FUNCTION_BLOCK FB_Fenster_Logik
VAR_IN_OUT
	Steuerung	: ST_Fenster_Steuerung;
	Zustand		: ST_Fenster_Zustand;
END_VAR
VAR_INPUT
	Parameter	: ST_Fenster_Parameter;
END_VAR
VAR_OUTPUT
END_VAR
VAR
END_VAR

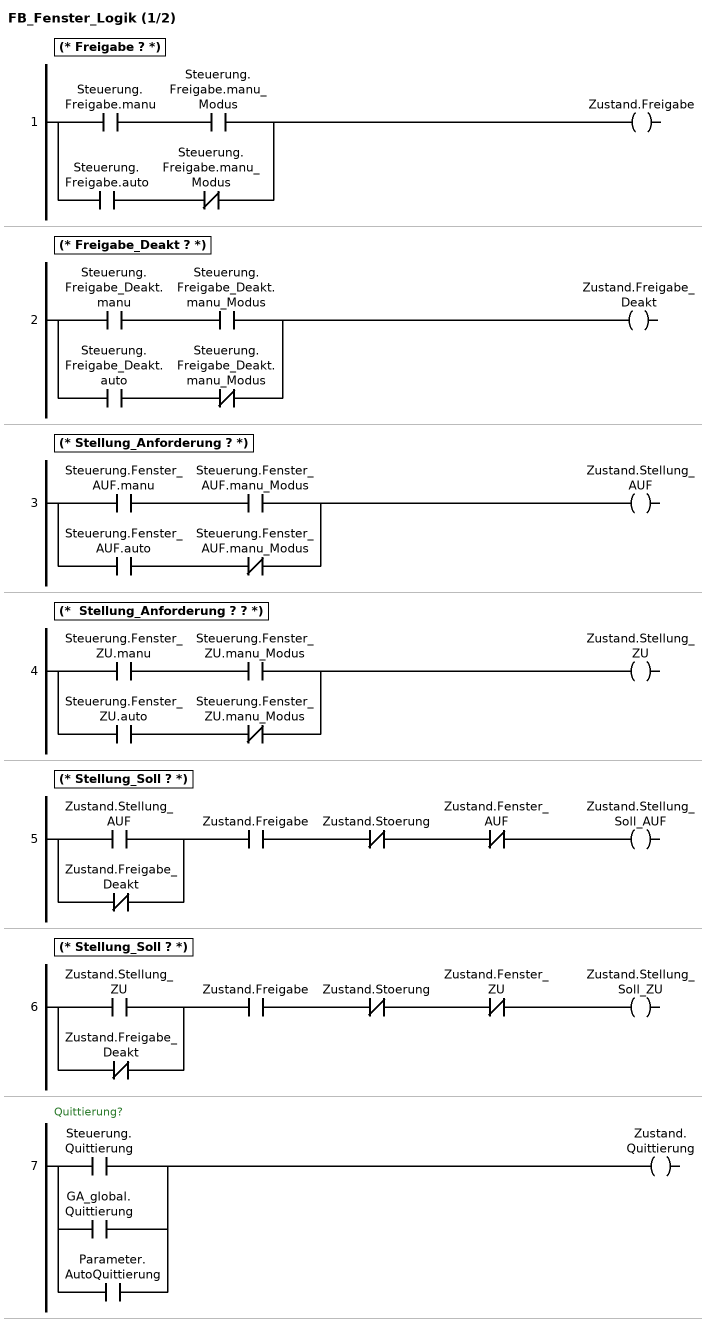
// NETWORK 1
// label: (* Freigabe ? *)
Zustand.Freigabe := Steuerung.Freigabe.manu AND Steuerung.Freigabe.manu_Modus OR Steuerung.Freigabe.auto AND NOT Steuerung.Freigabe.manu_Modus;

// NETWORK 2
// label: (* Freigabe_Deakt ? *)
Zustand.Freigabe_Deakt := Steuerung.Freigabe_Deakt.manu AND Steuerung.Freigabe_Deakt.manu_Modus OR Steuerung.Freigabe_Deakt.auto AND NOT Steuerung.Freigabe_Deakt.manu_Modus;

// NETWORK 3
// label: (* Stellung_Anforderung ? *)
Zustand.Stellung_AUF := Steuerung.Fenster_AUF.manu AND Steuerung.Fenster_AUF.manu_Modus OR Steuerung.Fenster_AUF.auto AND NOT Steuerung.Fenster_AUF.manu_Modus;

// NETWORK 4
// label: (*  Stellung_Anforderung ? ? *)
Zustand.Stellung_ZU := Steuerung.Fenster_ZU.manu AND Steuerung.Fenster_ZU.manu_Modus OR Steuerung.Fenster_ZU.auto AND NOT Steuerung.Fenster_ZU.manu_Modus;

// NETWORK 5
// label: (* Stellung_Soll ? *)
Zustand.Stellung_Soll_AUF := (Zustand.Stellung_AUF OR NOT Zustand.Freigabe_Deakt) AND Zustand.Freigabe AND NOT Zustand.Stoerung AND NOT Zustand.Fenster_AUF;

// NETWORK 6
// label: (* Stellung_Soll ? *)
Zustand.Stellung_Soll_ZU := (Zustand.Stellung_ZU OR NOT Zustand.Freigabe_Deakt) AND Zustand.Freigabe AND NOT Zustand.Stoerung AND NOT Zustand.Fenster_ZU;

// NETWORK 7
// Quittierung?
Zustand.Quittierung := Steuerung.Quittierung OR GA_global.Quittierung OR Parameter.AutoQuittierung;

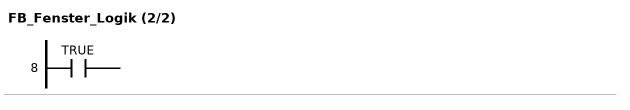
// NETWORK 8

END_FUNCTION_BLOCK

(* stored: Version 1.1.0.1, ProductVersion 3.1.4024.9
   POU FB_Fenster_Logik: Id {ce8ebaac-18d9-4eb4-87d7-dde0e2b43817}, SpecialFunc None *)
